INTERFACE ICommand EXTENDS IResult

PROPERTY Sequence : DINT
GET
END_GET
SET
END_SET
END_PROPERTY

METHOD Start : ICommand
VAR_INPUT
END_VAR
END_METHOD

END_INTERFACE

(* stored: Version 1.1.0.1, ProductVersion 3.1.4024.12
   Itf ICommand: Id {5865d299-3890-479b-b537-3d73a904f236}
   Property Sequence: Id {c401c39b-619e-4ccd-a272-221360d113f3}
   Get Get: Id {1d11e05b-d205-49a8-aa97-171585ecab97}
   Set Set: Id {5c7670eb-a3b6-4dff-84a1-325c18c4bb85}
   Method Start: Id {d2f31887-a413-4334-8bfa-3d772c5968bb} *)
